(* CoDeSys 2.3.9.47 project: NOT GATE.pro *)
(* Libraries: Nexgenie.lib 28.8.18 12:27:24, Standard.lib 28.8.18 12:27:25, Nexgenie_Util.lib 28.8.18 12:27:24, Nexgenie_H.lib 28.8.18 12:27:24, VAW.lib 28.8.18 12:27:25, Modbus.lib 28.8.18 12:27:24 *)

(* PLC configuration (modules and I/O channels)
Nexgenie1000 [Root] node -1, in %IB0 out %QB0
  Nexgenie [Nexgenie] node 0, in %IB0 out %QB0
*)

(* POU PLC_PRG, LD *)
PROGRAM PLC_PRG
VAR
	A AT %IX0.0: BOOL;
	Z AT %QX0.0: BOOL;
END_VAR
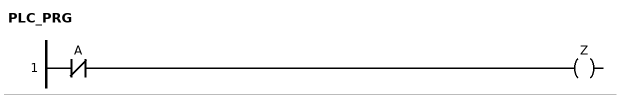
_LD_ (* Ladder Diagram *)
NETWORK 1
	[/A] --- (Z)
_END_LD_
(* the same logic as Structured Text *)
(* Network 1 *)
Z := NOT A;
END_PROGRAM

(* Visualisation LOL
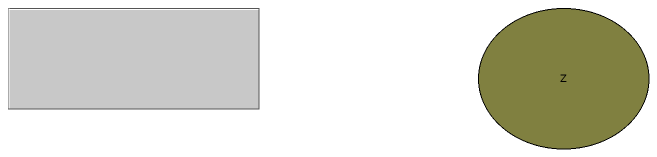
button at (90,70)-(341,171): toggles PLC_PRG.A
ellipse at (560,70)-(731,211): text "Z"; alarm colour if PLC_PRG.Z
*)
